// TIA Portal V17 export
// export: Created 2024-09-02T12:50:08.0346028Z, ExportSetting WithDefaults, DisplayName Totally Integrated Automation Portal, DisplayVersion V17, DisplayName TIA Portal Openness, DisplayVersion V17, DisplayName TIA Portal Version Control Interface, DisplayVersion V17, DisplayName STEP 7 Professional, DisplayVersion V17, DisplayName STEP 7 Safety, DisplayVersion V17, DisplayName WinCC Professional, DisplayVersion V17
FUNCTION "AnwFC1_FG02_Transport_OP70" : Void   // FC1381, LAD
TITLE = Transport
{ S7_Optimized_Access := 'TRUE' }
AUTHOR : VAF
FAMILY : SK
NAME : SK
VERSION : 0.1
// stored: AutoNumber false, IsIECCheckEnabled false, SetENOAutomatically false, UDAEnableTagReadback false
   VAR_TEMP
      Motion_Release : Bool;   // Bewegungsfreigabe / Motion permit
      Hand : Bool;
      Auto : Bool;
      t_ParityFault : Bool;
      t_ConfigFault : Bool;
      t_retval : Bool;
      "MM50/51_Home" : Bool;
      "MM50/51_Work" : Bool;
      "MM70/71_Home" : Bool;
      "MM70/71_Work" : Bool;
   END_VAR
BEGIN

REGION Network 1: Motion permit / Hand/ Auto / Bewegungsfreigabe / Hand / Auto
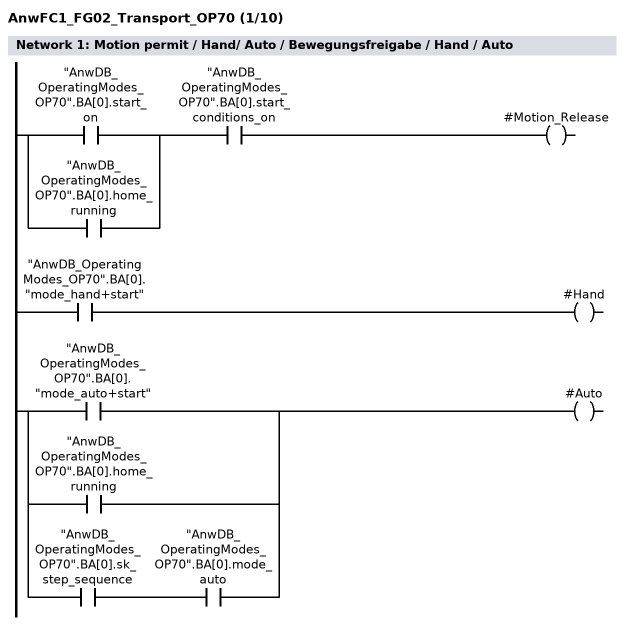
   RUNG wire#powerrail
      Contact( "AnwDB_OperatingModes_OP70".BA[0].start_on )
      wire#w1
      Contact( "AnwDB_OperatingModes_OP70".BA[0].start_conditions_on )
      Coil( #Motion_Release )
   END_RUNG
   RUNG wire#powerrail
      Contact( "AnwDB_OperatingModes_OP70".BA[0].home_running )
   END_RUNG wire#w1
   RUNG wire#powerrail
      Contact( "AnwDB_OperatingModes_OP70".BA[0]."mode_hand+start" )
      Coil( #Hand )
   END_RUNG
   RUNG wire#powerrail
      Contact( "AnwDB_OperatingModes_OP70".BA[0]."mode_auto+start" )
      wire#w2
      Coil( #Auto )
   END_RUNG
   RUNG wire#powerrail
      Contact( "AnwDB_OperatingModes_OP70".BA[0].home_running )
   END_RUNG wire#w2
   RUNG wire#powerrail
      Contact( "AnwDB_OperatingModes_OP70".BA[0].sk_step_sequence )
      Contact( "AnwDB_OperatingModes_OP70".BA[0].mode_auto )
   END_RUNG wire#w2
   // the same network as SCL:
   #Motion_Release := ("AnwDB_OperatingModes_OP70".BA[0].start_on OR "AnwDB_OperatingModes_OP70".BA[0].home_running) AND "AnwDB_OperatingModes_OP70".BA[0].start_conditions_on;
   #Hand := "AnwDB_OperatingModes_OP70".BA[0]."mode_hand+start";
   #Auto := "AnwDB_OperatingModes_OP70".BA[0]."mode_auto+start" OR "AnwDB_OperatingModes_OP70".BA[0].home_running OR ("AnwDB_OperatingModes_OP70".BA[0].sk_step_sequence AND "AnwDB_OperatingModes_OP70".BA[0].mode_auto);
END_REGION

REGION Network 2: Call of the step sequence / Aufruf der Schrittkette
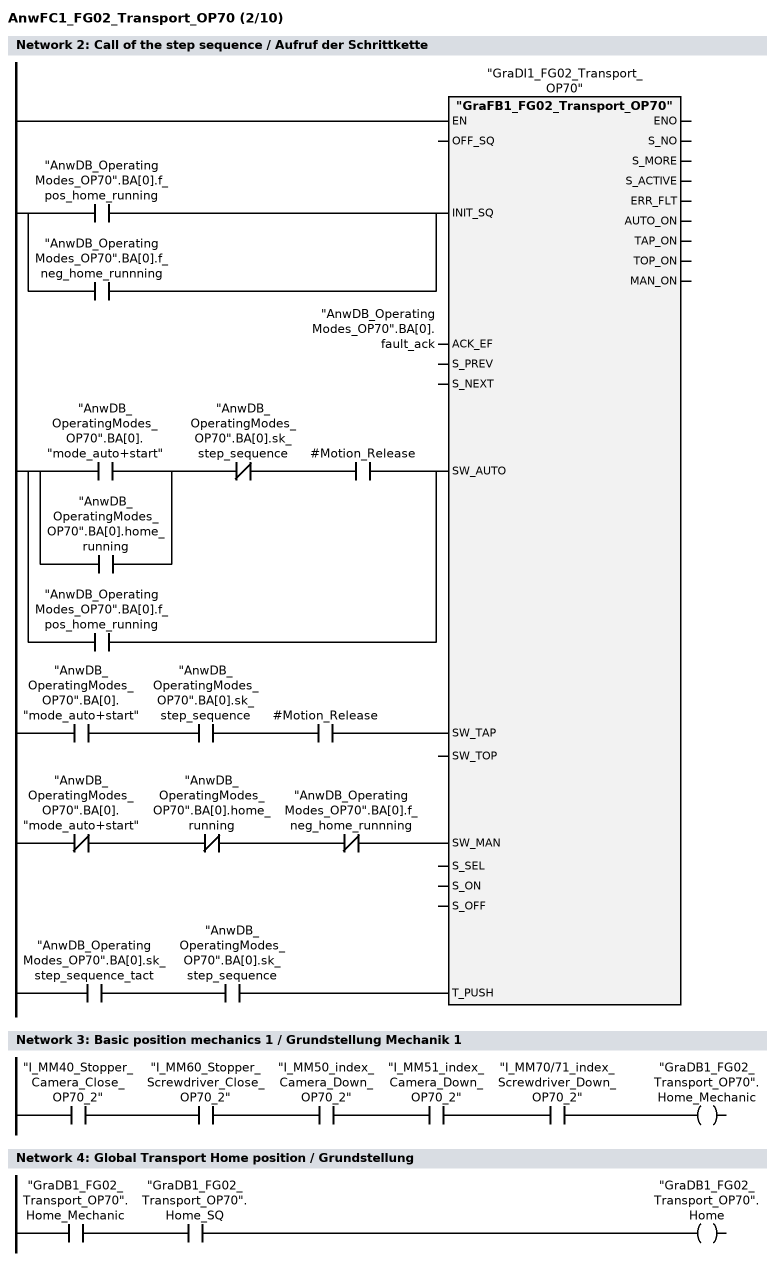
   RUNG wire#powerrail
      "GraDI1_FG02_Transport_OP70"(INIT_SQ := wire#w1, SW_AUTO := wire#w3, SW_TAP := wire#w4, SW_MAN := wire#w5, T_PUSH := wire#w6, OFF_SQ :=, ACK_EF := "AnwDB_OperatingModes_OP70".BA[0].fault_ack, S_PREV :=, S_NEXT :=, SW_TOP :=, S_SEL :=, S_ON :=, S_OFF :=, S_NO =>, S_MORE =>, S_ACTIVE =>, ERR_FLT =>, AUTO_ON =>, TAP_ON =>, TOP_ON =>, MAN_ON =>)
   END_RUNG
   RUNG wire#powerrail
      Contact( "AnwDB_OperatingModes_OP70".BA[0].f_pos_home_running )
   END_RUNG wire#w1
   RUNG wire#powerrail
      Contact( "AnwDB_OperatingModes_OP70".BA[0].f_neg_home_runnning )
   END_RUNG wire#w1
   RUNG wire#powerrail
      Contact( "AnwDB_OperatingModes_OP70".BA[0]."mode_auto+start" )
      wire#w2
      I_Contact( "AnwDB_OperatingModes_OP70".BA[0].sk_step_sequence )
      Contact( #Motion_Release )
   END_RUNG wire#w3
   RUNG wire#powerrail
      Contact( "AnwDB_OperatingModes_OP70".BA[0].home_running )
   END_RUNG wire#w2
   RUNG wire#powerrail
      Contact( "AnwDB_OperatingModes_OP70".BA[0].f_pos_home_running )
   END_RUNG wire#w3
   RUNG wire#powerrail
      Contact( "AnwDB_OperatingModes_OP70".BA[0]."mode_auto+start" )
      Contact( "AnwDB_OperatingModes_OP70".BA[0].sk_step_sequence )
      Contact( #Motion_Release )
   END_RUNG wire#w4
   RUNG wire#powerrail
      I_Contact( "AnwDB_OperatingModes_OP70".BA[0]."mode_auto+start" )
      I_Contact( "AnwDB_OperatingModes_OP70".BA[0].home_running )
      I_Contact( "AnwDB_OperatingModes_OP70".BA[0].f_neg_home_runnning )
   END_RUNG wire#w5
   RUNG wire#powerrail
      Contact( "AnwDB_OperatingModes_OP70".BA[0].sk_step_sequence_tact )
      Contact( "AnwDB_OperatingModes_OP70".BA[0].sk_step_sequence )
   END_RUNG wire#w6
   // the same network as SCL:
   "GraDI1_FG02_Transport_OP70"(INIT_SQ := "AnwDB_OperatingModes_OP70".BA[0].f_pos_home_running OR "AnwDB_OperatingModes_OP70".BA[0].f_neg_home_runnning,   // "GraFB1_FG02_Transport_OP70"
                           ACK_EF := "AnwDB_OperatingModes_OP70".BA[0].fault_ack,
                           SW_AUTO := (("AnwDB_OperatingModes_OP70".BA[0]."mode_auto+start" OR "AnwDB_OperatingModes_OP70".BA[0].home_running) AND NOT "AnwDB_OperatingModes_OP70".BA[0].sk_step_sequence AND #Motion_Release) OR "AnwDB_OperatingModes_OP70".BA[0].f_pos_home_running,
                           SW_TAP := "AnwDB_OperatingModes_OP70".BA[0]."mode_auto+start" AND "AnwDB_OperatingModes_OP70".BA[0].sk_step_sequence AND #Motion_Release,
                           SW_MAN := NOT "AnwDB_OperatingModes_OP70".BA[0]."mode_auto+start" AND NOT "AnwDB_OperatingModes_OP70".BA[0].home_running AND NOT "AnwDB_OperatingModes_OP70".BA[0].f_neg_home_runnning,
                           T_PUSH := "AnwDB_OperatingModes_OP70".BA[0].sk_step_sequence_tact AND "AnwDB_OperatingModes_OP70".BA[0].sk_step_sequence);
END_REGION

REGION Network 3: Basic position mechanics 1 / Grundstellung Mechanik 1
   RUNG wire#powerrail
      Contact( "I_MM40_Stopper_Camera_Close_OP70_2" )
      Contact( "I_MM60_Stopper_Screwdriver_Close_OP70_2" )
      Contact( "I_MM50_index_Camera_Down_OP70_2" )
      Contact( "I_MM51_index_Camera_Down_OP70_2" )
      Contact( "I_MM70/71_index_Screwdriver_Down_OP70_2" )
      Coil( "GraDB1_FG02_Transport_OP70".Home_Mechanic )
   END_RUNG
   // the same network as SCL:
   "GraDB1_FG02_Transport_OP70".Home_Mechanic := "I_MM40_Stopper_Camera_Close_OP70_2" AND "I_MM60_Stopper_Screwdriver_Close_OP70_2" AND "I_MM50_index_Camera_Down_OP70_2" AND "I_MM51_index_Camera_Down_OP70_2" AND "I_MM70/71_index_Screwdriver_Down_OP70_2";
END_REGION

REGION Network 4: Global Transport Home position / Grundstellung
   RUNG wire#powerrail
      Contact( "GraDB1_FG02_Transport_OP70".Home_Mechanic )
      Contact( "GraDB1_FG02_Transport_OP70".Home_SQ )
      Coil( "GraDB1_FG02_Transport_OP70".Home )
   END_RUNG
   // the same network as SCL:
   "GraDB1_FG02_Transport_OP70".Home := "GraDB1_FG02_Transport_OP70".Home_Mechanic AND "GraDB1_FG02_Transport_OP70".Home_SQ;
END_REGION

REGION Network 5: Finished message OK Camera / Fertigmeldung OK
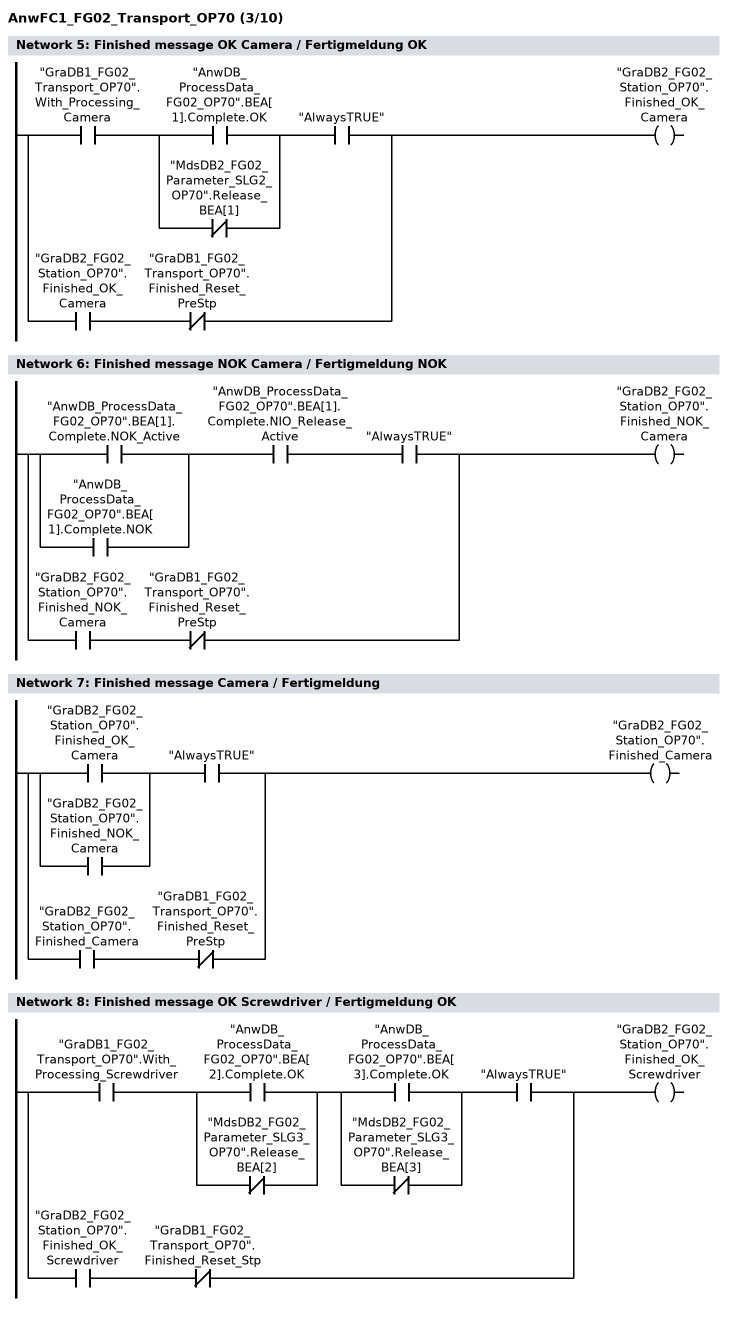
   RUNG wire#powerrail
      Contact( "GraDB1_FG02_Transport_OP70".With_Processing_Camera )
      wire#w1
      Contact( "AnwDB_ProcessData_FG02_OP70".BEA[1].Complete.OK )
      wire#w2
      Contact( "AlwaysTRUE" )
      wire#w3
      Coil( "GraDB2_FG02_Station_OP70".Finished_OK_Camera )
   END_RUNG
   RUNG wire#w1
      I_Contact( "MdsDB2_FG02_Parameter_SLG2_OP70".Release_BEA[1] )
   END_RUNG wire#w2
   RUNG wire#powerrail
      Contact( "GraDB2_FG02_Station_OP70".Finished_OK_Camera )
      I_Contact( "GraDB1_FG02_Transport_OP70".Finished_Reset_PreStp )
   END_RUNG wire#w3
   // the same network as SCL:
   "GraDB2_FG02_Station_OP70".Finished_OK_Camera := ("GraDB1_FG02_Transport_OP70".With_Processing_Camera AND ("AnwDB_ProcessData_FG02_OP70".BEA[1].Complete.OK OR NOT "MdsDB2_FG02_Parameter_SLG2_OP70".Release_BEA[1]) AND "AlwaysTRUE") OR ("GraDB2_FG02_Station_OP70".Finished_OK_Camera AND NOT "GraDB1_FG02_Transport_OP70".Finished_Reset_PreStp);
END_REGION

REGION Network 6: Finished message NOK Camera / Fertigmeldung NOK
   RUNG wire#powerrail
      Contact( "AnwDB_ProcessData_FG02_OP70".BEA[1].Complete.NOK_Active )
      wire#w1
      Contact( "AnwDB_ProcessData_FG02_OP70".BEA[1].Complete.NIO_Release_Active )
      Contact( "AlwaysTRUE" )
      wire#w2
      Coil( "GraDB2_FG02_Station_OP70".Finished_NOK_Camera )
   END_RUNG
   RUNG wire#powerrail
      Contact( "AnwDB_ProcessData_FG02_OP70".BEA[1].Complete.NOK )
   END_RUNG wire#w1
   RUNG wire#powerrail
      Contact( "GraDB2_FG02_Station_OP70".Finished_NOK_Camera )
      I_Contact( "GraDB1_FG02_Transport_OP70".Finished_Reset_PreStp )
   END_RUNG wire#w2
   // the same network as SCL:
   "GraDB2_FG02_Station_OP70".Finished_NOK_Camera := (("AnwDB_ProcessData_FG02_OP70".BEA[1].Complete.NOK_Active OR "AnwDB_ProcessData_FG02_OP70".BEA[1].Complete.NOK) AND "AnwDB_ProcessData_FG02_OP70".BEA[1].Complete.NIO_Release_Active AND "AlwaysTRUE") OR ("GraDB2_FG02_Station_OP70".Finished_NOK_Camera AND NOT "GraDB1_FG02_Transport_OP70".Finished_Reset_PreStp);
END_REGION

REGION Network 7: Finished message Camera / Fertigmeldung
   RUNG wire#powerrail
      Contact( "GraDB2_FG02_Station_OP70".Finished_OK_Camera )
      wire#w1
      Contact( "AlwaysTRUE" )
      wire#w2
      Coil( "GraDB2_FG02_Station_OP70".Finished_Camera )
   END_RUNG
   RUNG wire#powerrail
      Contact( "GraDB2_FG02_Station_OP70".Finished_NOK_Camera )
   END_RUNG wire#w1
   RUNG wire#powerrail
      Contact( "GraDB2_FG02_Station_OP70".Finished_Camera )
      I_Contact( "GraDB1_FG02_Transport_OP70".Finished_Reset_PreStp )
   END_RUNG wire#w2
   // the same network as SCL:
   "GraDB2_FG02_Station_OP70".Finished_Camera := (("GraDB2_FG02_Station_OP70".Finished_OK_Camera OR "GraDB2_FG02_Station_OP70".Finished_NOK_Camera) AND "AlwaysTRUE") OR ("GraDB2_FG02_Station_OP70".Finished_Camera AND NOT "GraDB1_FG02_Transport_OP70".Finished_Reset_PreStp);
END_REGION

REGION Network 8: Finished message OK Screwdriver / Fertigmeldung OK
   RUNG wire#powerrail
      Contact( "GraDB1_FG02_Transport_OP70".With_Processing_Screwdriver )
      wire#w1
      Contact( "AnwDB_ProcessData_FG02_OP70".BEA[2].Complete.OK )
      wire#w2
      Contact( "AnwDB_ProcessData_FG02_OP70".BEA[3].Complete.OK )
      wire#w3
      Contact( "AlwaysTRUE" )
      wire#w4
      Coil( "GraDB2_FG02_Station_OP70".Finished_OK_Screwdriver )
   END_RUNG
   RUNG wire#w1
      I_Contact( "MdsDB2_FG02_Parameter_SLG3_OP70".Release_BEA[2] )
   END_RUNG wire#w2
   RUNG wire#w2
      I_Contact( "MdsDB2_FG02_Parameter_SLG3_OP70".Release_BEA[3] )
   END_RUNG wire#w3
   RUNG wire#powerrail
      Contact( "GraDB2_FG02_Station_OP70".Finished_OK_Screwdriver )
      I_Contact( "GraDB1_FG02_Transport_OP70".Finished_Reset_Stp )
   END_RUNG wire#w4
   // the same network as SCL:
   "GraDB2_FG02_Station_OP70".Finished_OK_Screwdriver := ("GraDB1_FG02_Transport_OP70".With_Processing_Screwdriver AND ("AnwDB_ProcessData_FG02_OP70".BEA[2].Complete.OK OR NOT "MdsDB2_FG02_Parameter_SLG3_OP70".Release_BEA[2]) AND ("AnwDB_ProcessData_FG02_OP70".BEA[3].Complete.OK OR NOT "MdsDB2_FG02_Parameter_SLG3_OP70".Release_BEA[3]) AND "AlwaysTRUE") OR ("GraDB2_FG02_Station_OP70".Finished_OK_Screwdriver AND NOT "GraDB1_FG02_Transport_OP70".Finished_Reset_Stp);
END_REGION

REGION Network 9: Finished message NOK Screwdriver / Fertigmeldung NOK
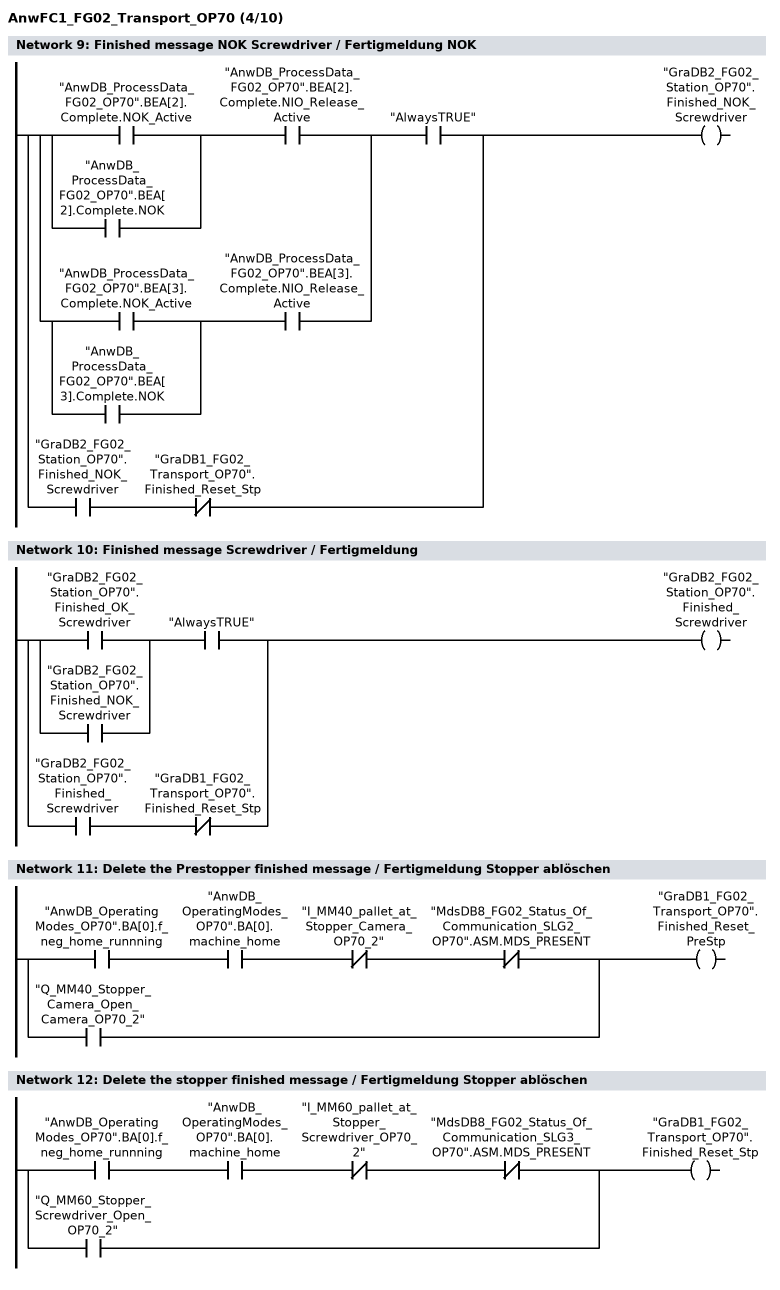
   RUNG wire#powerrail
      Contact( "AnwDB_ProcessData_FG02_OP70".BEA[2].Complete.NOK_Active )
      wire#w1
      Contact( "AnwDB_ProcessData_FG02_OP70".BEA[2].Complete.NIO_Release_Active )
      wire#w2
      Contact( "AlwaysTRUE" )
      wire#w4
      Coil( "GraDB2_FG02_Station_OP70".Finished_NOK_Screwdriver )
   END_RUNG
   RUNG wire#powerrail
      Contact( "AnwDB_ProcessData_FG02_OP70".BEA[2].Complete.NOK )
   END_RUNG wire#w1
   RUNG wire#powerrail
      Contact( "AnwDB_ProcessData_FG02_OP70".BEA[3].Complete.NOK_Active )
      wire#w3
      Contact( "AnwDB_ProcessData_FG02_OP70".BEA[3].Complete.NIO_Release_Active )
   END_RUNG wire#w2
   RUNG wire#powerrail
      Contact( "AnwDB_ProcessData_FG02_OP70".BEA[3].Complete.NOK )
   END_RUNG wire#w3
   RUNG wire#powerrail
      Contact( "GraDB2_FG02_Station_OP70".Finished_NOK_Screwdriver )
      I_Contact( "GraDB1_FG02_Transport_OP70".Finished_Reset_Stp )
   END_RUNG wire#w4
   // the same network as SCL:
   "GraDB2_FG02_Station_OP70".Finished_NOK_Screwdriver := (((("AnwDB_ProcessData_FG02_OP70".BEA[2].Complete.NOK_Active OR "AnwDB_ProcessData_FG02_OP70".BEA[2].Complete.NOK) AND "AnwDB_ProcessData_FG02_OP70".BEA[2].Complete.NIO_Release_Active) OR (("AnwDB_ProcessData_FG02_OP70".BEA[3].Complete.NOK_Active OR "AnwDB_ProcessData_FG02_OP70".BEA[3].Complete.NOK) AND "AnwDB_ProcessData_FG02_OP70".BEA[3].Complete.NIO_Release_Active)) AND "AlwaysTRUE") OR ("GraDB2_FG02_Station_OP70".Finished_NOK_Screwdriver AND NOT "GraDB1_FG02_Transport_OP70".Finished_Reset_Stp);
END_REGION

REGION Network 10: Finished message Screwdriver / Fertigmeldung
   RUNG wire#powerrail
      Contact( "GraDB2_FG02_Station_OP70".Finished_OK_Screwdriver )
      wire#w1
      Contact( "AlwaysTRUE" )
      wire#w2
      Coil( "GraDB2_FG02_Station_OP70".Finished_Screwdriver )
   END_RUNG
   RUNG wire#powerrail
      Contact( "GraDB2_FG02_Station_OP70".Finished_NOK_Screwdriver )
   END_RUNG wire#w1
   RUNG wire#powerrail
      Contact( "GraDB2_FG02_Station_OP70".Finished_Screwdriver )
      I_Contact( "GraDB1_FG02_Transport_OP70".Finished_Reset_Stp )
   END_RUNG wire#w2
   // the same network as SCL:
   "GraDB2_FG02_Station_OP70".Finished_Screwdriver := (("GraDB2_FG02_Station_OP70".Finished_OK_Screwdriver OR "GraDB2_FG02_Station_OP70".Finished_NOK_Screwdriver) AND "AlwaysTRUE") OR ("GraDB2_FG02_Station_OP70".Finished_Screwdriver AND NOT "GraDB1_FG02_Transport_OP70".Finished_Reset_Stp);
END_REGION

REGION Network 11: Delete the Prestopper finished message / Fertigmeldung Stopper ablöschen
   RUNG wire#powerrail
      Contact( "AnwDB_OperatingModes_OP70".BA[0].f_neg_home_runnning )
      Contact( "AnwDB_OperatingModes_OP70".BA[0].machine_home )
      I_Contact( "I_MM40_pallet_at_Stopper_Camera_OP70_2" )
      I_Contact( "MdsDB8_FG02_Status_Of_Communication_SLG2_OP70".ASM.MDS_PRESENT )
      wire#w1
      Coil( "GraDB1_FG02_Transport_OP70".Finished_Reset_PreStp )
   END_RUNG
   RUNG wire#powerrail
      Contact( "Q_MM40_Stopper_Camera_Open_Camera_OP70_2" )
   END_RUNG wire#w1
   // the same network as SCL:
   "GraDB1_FG02_Transport_OP70".Finished_Reset_PreStp := ("AnwDB_OperatingModes_OP70".BA[0].f_neg_home_runnning AND "AnwDB_OperatingModes_OP70".BA[0].machine_home AND NOT "I_MM40_pallet_at_Stopper_Camera_OP70_2" AND NOT "MdsDB8_FG02_Status_Of_Communication_SLG2_OP70".ASM.MDS_PRESENT) OR "Q_MM40_Stopper_Camera_Open_Camera_OP70_2";
END_REGION

REGION Network 12: Delete the stopper finished message / Fertigmeldung Stopper ablöschen
   RUNG wire#powerrail
      Contact( "AnwDB_OperatingModes_OP70".BA[0].f_neg_home_runnning )
      Contact( "AnwDB_OperatingModes_OP70".BA[0].machine_home )
      I_Contact( "I_MM60_pallet_at_Stopper_Screwdriver_OP70_2" )
      I_Contact( "MdsDB8_FG02_Status_Of_Communication_SLG3_OP70".ASM.MDS_PRESENT )
      wire#w1
      Coil( "GraDB1_FG02_Transport_OP70".Finished_Reset_Stp )
   END_RUNG
   RUNG wire#powerrail
      Contact( "Q_MM60_Stopper_Screwdriver_Open_OP70_2" )
   END_RUNG wire#w1
   // the same network as SCL:
   "GraDB1_FG02_Transport_OP70".Finished_Reset_Stp := ("AnwDB_OperatingModes_OP70".BA[0].f_neg_home_runnning AND "AnwDB_OperatingModes_OP70".BA[0].machine_home AND NOT "I_MM60_pallet_at_Stopper_Screwdriver_OP70_2" AND NOT "MdsDB8_FG02_Status_Of_Communication_SLG3_OP70".ASM.MDS_PRESENT) OR "Q_MM60_Stopper_Screwdriver_Open_OP70_2";
END_REGION

REGION Network 13: WT in Station
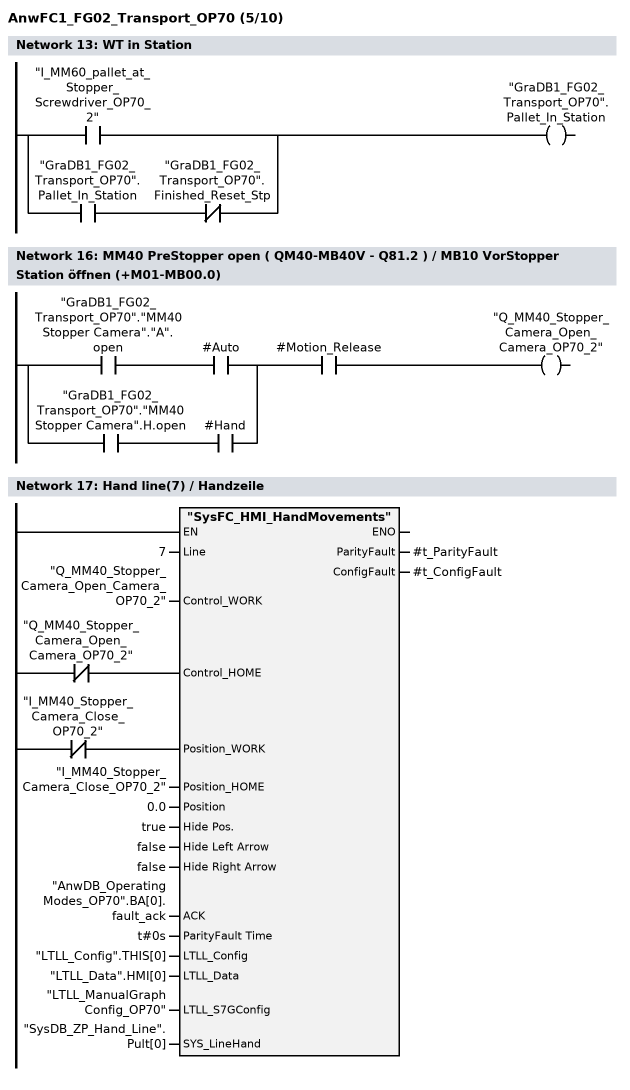
   RUNG wire#powerrail
      Contact( "I_MM60_pallet_at_Stopper_Screwdriver_OP70_2" )
      wire#w1
      Coil( "GraDB1_FG02_Transport_OP70".Pallet_In_Station )
   END_RUNG
   RUNG wire#powerrail
      Contact( "GraDB1_FG02_Transport_OP70".Pallet_In_Station )
      I_Contact( "GraDB1_FG02_Transport_OP70".Finished_Reset_Stp )
   END_RUNG wire#w1
   // the same network as SCL:
   "GraDB1_FG02_Transport_OP70".Pallet_In_Station := "I_MM60_pallet_at_Stopper_Screwdriver_OP70_2" OR ("GraDB1_FG02_Transport_OP70".Pallet_In_Station AND NOT "GraDB1_FG02_Transport_OP70".Finished_Reset_Stp);
END_REGION

REGION Network 14: ########### USER ########### / ########### ANWENDER ###########
END_REGION

REGION Network 15: ########### SS_02_001_Setup ###########
END_REGION

REGION Network 16: MM40 PreStopper open ( QM40-MB40V - Q81.2 ) / MB10 VorStopper Station öffnen (+M01-MB00.0)
   RUNG wire#powerrail
      Contact( "GraDB1_FG02_Transport_OP70"."MM40 Stopper Camera"."A".open )
      Contact( #Auto )
      wire#w1
      Contact( #Motion_Release )
      Coil( "Q_MM40_Stopper_Camera_Open_Camera_OP70_2" )
   END_RUNG
   RUNG wire#powerrail
      Contact( "GraDB1_FG02_Transport_OP70"."MM40 Stopper Camera".H.open )
      Contact( #Hand )
   END_RUNG wire#w1
   // the same network as SCL:
   "Q_MM40_Stopper_Camera_Open_Camera_OP70_2" := (("GraDB1_FG02_Transport_OP70"."MM40 Stopper Camera"."A".open AND #Auto) OR ("GraDB1_FG02_Transport_OP70"."MM40 Stopper Camera".H.open AND #Hand)) AND #Motion_Release;
END_REGION

REGION Network 17: Hand line(7) / Handzeile
   RUNG wire#powerrail
      "SysFC_HMI_HandMovements"(Control_HOME := wire#w1, Position_WORK := wire#w2, Line := 7, Control_WORK := "Q_MM40_Stopper_Camera_Open_Camera_OP70_2", Position_HOME := "I_MM40_Stopper_Camera_Close_OP70_2", Position := 0.0, "Hide Pos." := true, "Hide Left Arrow" := false, "Hide Right Arrow" := false, ACK := "AnwDB_OperatingModes_OP70".BA[0].fault_ack, "ParityFault Time" := t#0s, LTLL_Config := "LTLL_Config".THIS[0], LTLL_Data := "LTLL_Data".HMI[0], LTLL_S7GConfig := "LTLL_ManualGraphConfig_OP70", SYS_LineHand := "SysDB_ZP_Hand_Line".Pult[0], ParityFault => #t_ParityFault, ConfigFault => #t_ConfigFault)
   END_RUNG
   RUNG wire#powerrail
      I_Contact( "Q_MM40_Stopper_Camera_Open_Camera_OP70_2" )
   END_RUNG wire#w1
   RUNG wire#powerrail
      I_Contact( "I_MM40_Stopper_Camera_Close_OP70_2" )
   END_RUNG wire#w2
   // the same network as SCL:
   "SysFC_HMI_HandMovements"(Line := 7,
                           Control_WORK := "Q_MM40_Stopper_Camera_Open_Camera_OP70_2",
                           Control_HOME := NOT "Q_MM40_Stopper_Camera_Open_Camera_OP70_2",
                           Position_WORK := NOT "I_MM40_Stopper_Camera_Close_OP70_2",
                           Position_HOME := "I_MM40_Stopper_Camera_Close_OP70_2",
                           Position := 0.0,
                           "Hide Pos." := true,
                           "Hide Left Arrow" := false,
                           "Hide Right Arrow" := false,
                           ACK := "AnwDB_OperatingModes_OP70".BA[0].fault_ack,
                           "ParityFault Time" := t#0s,
                           LTLL_Config := "LTLL_Config".THIS[0],
                           LTLL_Data := "LTLL_Data".HMI[0],
                           LTLL_S7GConfig := "LTLL_ManualGraphConfig_OP70",
                           SYS_LineHand := "SysDB_ZP_Hand_Line".Pult[0],
                           ParityFault => #t_ParityFault,
                           ConfigFault => #t_ConfigFault);
END_REGION

REGION Network 18: Hand line SLG2 Prestopper read / write (8) / SLG BX600 schreiben / lesen
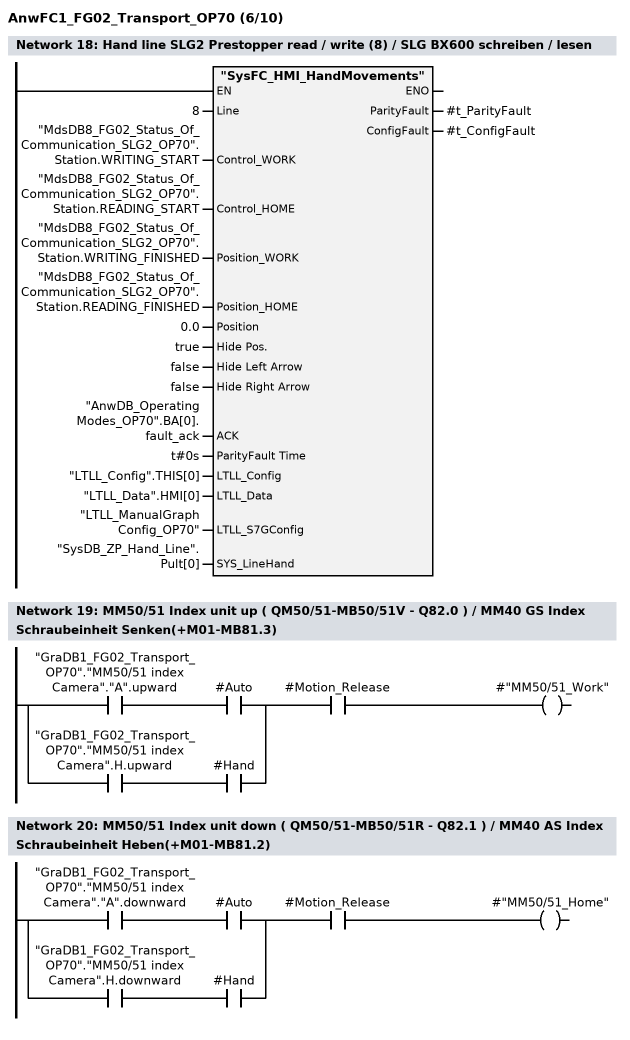
   RUNG wire#powerrail
      "SysFC_HMI_HandMovements"(Line := 8, Control_WORK := "MdsDB8_FG02_Status_Of_Communication_SLG2_OP70".Station.WRITING_START, Control_HOME := "MdsDB8_FG02_Status_Of_Communication_SLG2_OP70".Station.READING_START, Position_WORK := "MdsDB8_FG02_Status_Of_Communication_SLG2_OP70".Station.WRITING_FINISHED, Position_HOME := "MdsDB8_FG02_Status_Of_Communication_SLG2_OP70".Station.READING_FINISHED, Position := 0.0, "Hide Pos." := true, "Hide Left Arrow" := false, "Hide Right Arrow" := false, ACK := "AnwDB_OperatingModes_OP70".BA[0].fault_ack, "ParityFault Time" := t#0s, LTLL_Config := "LTLL_Config".THIS[0], LTLL_Data := "LTLL_Data".HMI[0], LTLL_S7GConfig := "LTLL_ManualGraphConfig_OP70", SYS_LineHand := "SysDB_ZP_Hand_Line".Pult[0], ParityFault => #t_ParityFault, ConfigFault => #t_ConfigFault)
   END_RUNG
   // the same network as SCL:
   "SysFC_HMI_HandMovements"(Line := 8,
                           Control_WORK := "MdsDB8_FG02_Status_Of_Communication_SLG2_OP70".Station.WRITING_START,
                           Control_HOME := "MdsDB8_FG02_Status_Of_Communication_SLG2_OP70".Station.READING_START,
                           Position_WORK := "MdsDB8_FG02_Status_Of_Communication_SLG2_OP70".Station.WRITING_FINISHED,
                           Position_HOME := "MdsDB8_FG02_Status_Of_Communication_SLG2_OP70".Station.READING_FINISHED,
                           Position := 0.0,
                           "Hide Pos." := true,
                           "Hide Left Arrow" := false,
                           "Hide Right Arrow" := false,
                           ACK := "AnwDB_OperatingModes_OP70".BA[0].fault_ack,
                           "ParityFault Time" := t#0s,
                           LTLL_Config := "LTLL_Config".THIS[0],
                           LTLL_Data := "LTLL_Data".HMI[0],
                           LTLL_S7GConfig := "LTLL_ManualGraphConfig_OP70",
                           SYS_LineHand := "SysDB_ZP_Hand_Line".Pult[0],
                           ParityFault => #t_ParityFault,
                           ConfigFault => #t_ConfigFault);
END_REGION

REGION Network 19: MM50/51 Index unit up ( QM50/51-MB50/51V - Q82.0 ) / MM40 GS Index Schraubeinheit Senken(+M01-MB81.3)
   RUNG wire#powerrail
      Contact( "GraDB1_FG02_Transport_OP70"."MM50/51 index Camera"."A".upward )
      Contact( #Auto )
      wire#w1
      Contact( #Motion_Release )
      Coil( #"MM50/51_Work" )
   END_RUNG
   RUNG wire#powerrail
      Contact( "GraDB1_FG02_Transport_OP70"."MM50/51 index Camera".H.upward )
      Contact( #Hand )
   END_RUNG wire#w1
   // the same network as SCL:
   #"MM50/51_Work" := (("GraDB1_FG02_Transport_OP70"."MM50/51 index Camera"."A".upward AND #Auto) OR ("GraDB1_FG02_Transport_OP70"."MM50/51 index Camera".H.upward AND #Hand)) AND #Motion_Release;
END_REGION

REGION Network 20: MM50/51 Index unit down ( QM50/51-MB50/51R - Q82.1 ) / MM40 AS Index Schraubeinheit Heben(+M01-MB81.2)
   RUNG wire#powerrail
      Contact( "GraDB1_FG02_Transport_OP70"."MM50/51 index Camera"."A".downward )
      Contact( #Auto )
      wire#w1
      Contact( #Motion_Release )
      Coil( #"MM50/51_Home" )
   END_RUNG
   RUNG wire#powerrail
      Contact( "GraDB1_FG02_Transport_OP70"."MM50/51 index Camera".H.downward )
      Contact( #Hand )
   END_RUNG wire#w1
   // the same network as SCL:
   #"MM50/51_Home" := (("GraDB1_FG02_Transport_OP70"."MM50/51 index Camera"."A".downward AND #Auto) OR ("GraDB1_FG02_Transport_OP70"."MM50/51 index Camera".H.downward AND #Hand)) AND #Motion_Release;
END_REGION

REGION Network 21: HLP - Index Up/Down / MM40 - HLP Pneumatik
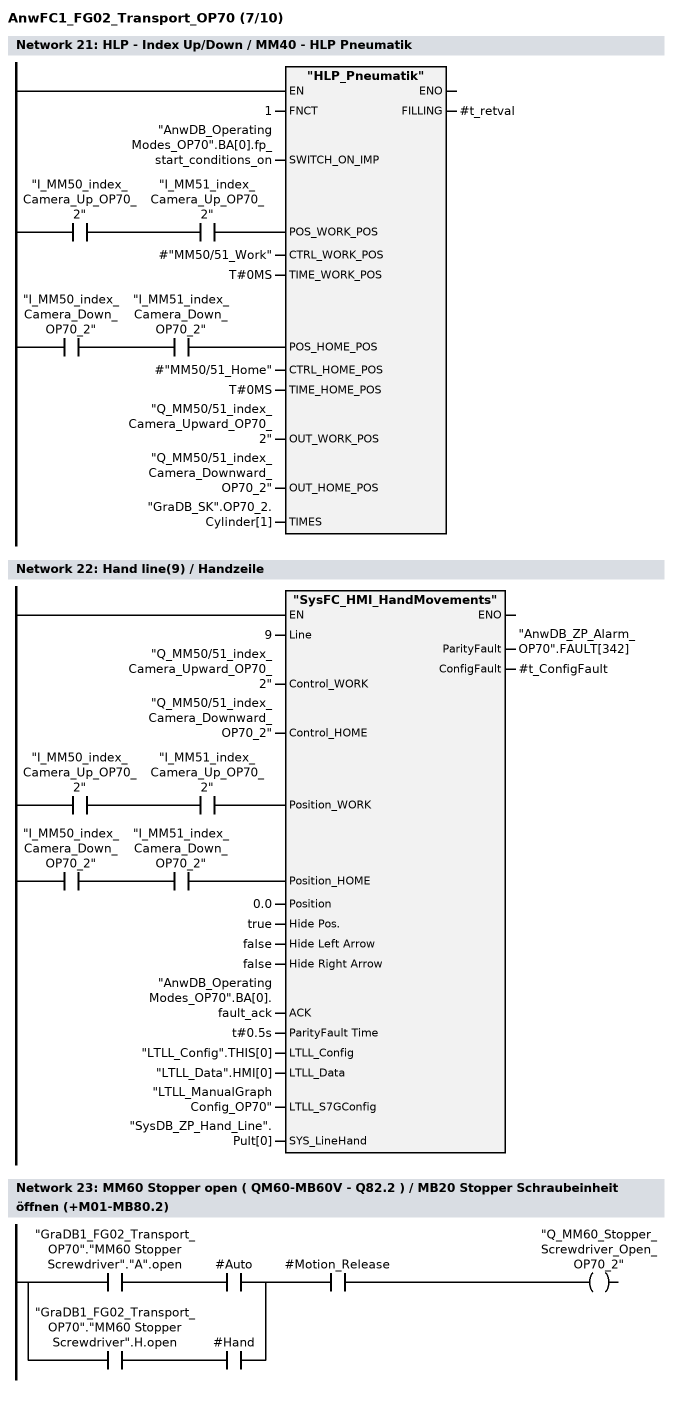
   RUNG wire#powerrail
      "HLP_Pneumatik"(POS_WORK_POS := wire#w1, POS_HOME_POS := wire#w2, FNCT := 1, SWITCH_ON_IMP := "AnwDB_OperatingModes_OP70".BA[0].fp_start_conditions_on, CTRL_WORK_POS := #"MM50/51_Work", TIME_WORK_POS := T#0MS, CTRL_HOME_POS := #"MM50/51_Home", TIME_HOME_POS := T#0MS, OUT_WORK_POS := "Q_MM50/51_index_Camera_Upward_OP70_2", OUT_HOME_POS := "Q_MM50/51_index_Camera_Downward_OP70_2", TIMES := "GraDB_SK".OP70_2.Cylinder[1], FILLING => #t_retval)
   END_RUNG
   RUNG wire#powerrail
      Contact( "I_MM50_index_Camera_Up_OP70_2" )
      Contact( "I_MM51_index_Camera_Up_OP70_2" )
   END_RUNG wire#w1
   RUNG wire#powerrail
      Contact( "I_MM50_index_Camera_Down_OP70_2" )
      Contact( "I_MM51_index_Camera_Down_OP70_2" )
   END_RUNG wire#w2
   // the same network as SCL:
   "HLP_Pneumatik"(FNCT := 1,
                   SWITCH_ON_IMP := "AnwDB_OperatingModes_OP70".BA[0].fp_start_conditions_on,
                   POS_WORK_POS := "I_MM50_index_Camera_Up_OP70_2" AND "I_MM51_index_Camera_Up_OP70_2",
                   CTRL_WORK_POS := #"MM50/51_Work",
                   TIME_WORK_POS := T#0MS,
                   POS_HOME_POS := "I_MM50_index_Camera_Down_OP70_2" AND "I_MM51_index_Camera_Down_OP70_2",
                   CTRL_HOME_POS := #"MM50/51_Home",
                   TIME_HOME_POS := T#0MS,
                   OUT_WORK_POS := "Q_MM50/51_index_Camera_Upward_OP70_2",
                   OUT_HOME_POS := "Q_MM50/51_index_Camera_Downward_OP70_2",
                   TIMES := "GraDB_SK".OP70_2.Cylinder[1],
                   FILLING => #t_retval);
END_REGION

REGION Network 22: Hand line(9) / Handzeile
   RUNG wire#powerrail
      "SysFC_HMI_HandMovements"(Position_WORK := wire#w1, Position_HOME := wire#w2, Line := 9, Control_WORK := "Q_MM50/51_index_Camera_Upward_OP70_2", Control_HOME := "Q_MM50/51_index_Camera_Downward_OP70_2", Position := 0.0, "Hide Pos." := true, "Hide Left Arrow" := false, "Hide Right Arrow" := false, ACK := "AnwDB_OperatingModes_OP70".BA[0].fault_ack, "ParityFault Time" := t#0.5s, LTLL_Config := "LTLL_Config".THIS[0], LTLL_Data := "LTLL_Data".HMI[0], LTLL_S7GConfig := "LTLL_ManualGraphConfig_OP70", SYS_LineHand := "SysDB_ZP_Hand_Line".Pult[0], ParityFault => "AnwDB_ZP_Alarm_OP70".FAULT[342], ConfigFault => #t_ConfigFault)
   END_RUNG
   RUNG wire#powerrail
      Contact( "I_MM50_index_Camera_Up_OP70_2" )
      Contact( "I_MM51_index_Camera_Up_OP70_2" )
   END_RUNG wire#w1
   RUNG wire#powerrail
      Contact( "I_MM50_index_Camera_Down_OP70_2" )
      Contact( "I_MM51_index_Camera_Down_OP70_2" )
   END_RUNG wire#w2
   // the same network as SCL:
   "SysFC_HMI_HandMovements"(Line := 9,
                           Control_WORK := "Q_MM50/51_index_Camera_Upward_OP70_2",
                           Control_HOME := "Q_MM50/51_index_Camera_Downward_OP70_2",
                           Position_WORK := "I_MM50_index_Camera_Up_OP70_2" AND "I_MM51_index_Camera_Up_OP70_2",
                           Position_HOME := "I_MM50_index_Camera_Down_OP70_2" AND "I_MM51_index_Camera_Down_OP70_2",
                           Position := 0.0,
                           "Hide Pos." := true,
                           "Hide Left Arrow" := false,
                           "Hide Right Arrow" := false,
                           ACK := "AnwDB_OperatingModes_OP70".BA[0].fault_ack,
                           "ParityFault Time" := t#0.5s,
                           LTLL_Config := "LTLL_Config".THIS[0],
                           LTLL_Data := "LTLL_Data".HMI[0],
                           LTLL_S7GConfig := "LTLL_ManualGraphConfig_OP70",
                           SYS_LineHand := "SysDB_ZP_Hand_Line".Pult[0],
                           ParityFault => "AnwDB_ZP_Alarm_OP70".FAULT[342],
                           ConfigFault => #t_ConfigFault);
END_REGION

REGION Network 23: MM60 Stopper open ( QM60-MB60V - Q82.2 ) / MB20 Stopper Schraubeinheit öffnen (+M01-MB80.2)
   RUNG wire#powerrail
      Contact( "GraDB1_FG02_Transport_OP70"."MM60 Stopper Screwdriver"."A".open )
      Contact( #Auto )
      wire#w1
      Contact( #Motion_Release )
      Coil( "Q_MM60_Stopper_Screwdriver_Open_OP70_2" )
   END_RUNG
   RUNG wire#powerrail
      Contact( "GraDB1_FG02_Transport_OP70"."MM60 Stopper Screwdriver".H.open )
      Contact( #Hand )
   END_RUNG wire#w1
   // the same network as SCL:
   "Q_MM60_Stopper_Screwdriver_Open_OP70_2" := (("GraDB1_FG02_Transport_OP70"."MM60 Stopper Screwdriver"."A".open AND #Auto) OR ("GraDB1_FG02_Transport_OP70"."MM60 Stopper Screwdriver".H.open AND #Hand)) AND #Motion_Release;
END_REGION

REGION Network 24: Hand line(10) / Handzeile
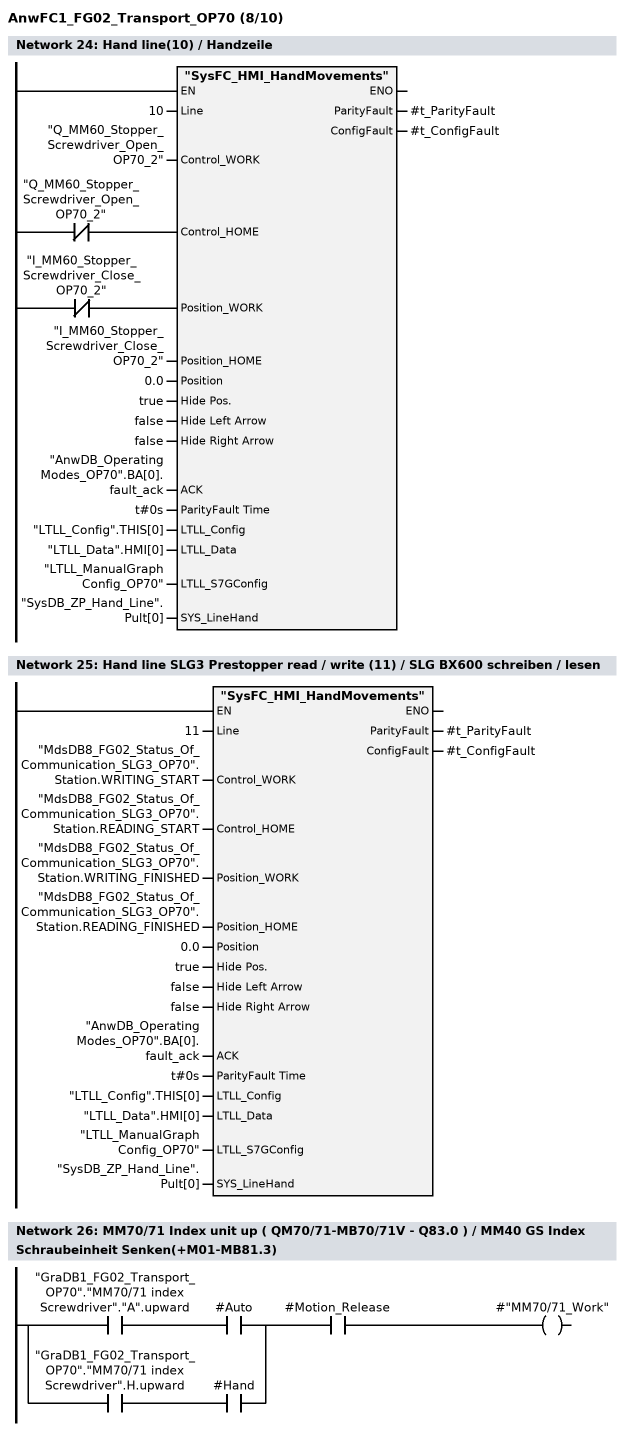
   RUNG wire#powerrail
      "SysFC_HMI_HandMovements"(Control_HOME := wire#w1, Position_WORK := wire#w2, Line := 10, Control_WORK := "Q_MM60_Stopper_Screwdriver_Open_OP70_2", Position_HOME := "I_MM60_Stopper_Screwdriver_Close_OP70_2", Position := 0.0, "Hide Pos." := true, "Hide Left Arrow" := false, "Hide Right Arrow" := false, ACK := "AnwDB_OperatingModes_OP70".BA[0].fault_ack, "ParityFault Time" := t#0s, LTLL_Config := "LTLL_Config".THIS[0], LTLL_Data := "LTLL_Data".HMI[0], LTLL_S7GConfig := "LTLL_ManualGraphConfig_OP70", SYS_LineHand := "SysDB_ZP_Hand_Line".Pult[0], ParityFault => #t_ParityFault, ConfigFault => #t_ConfigFault)
   END_RUNG
   RUNG wire#powerrail
      I_Contact( "Q_MM60_Stopper_Screwdriver_Open_OP70_2" )
   END_RUNG wire#w1
   RUNG wire#powerrail
      I_Contact( "I_MM60_Stopper_Screwdriver_Close_OP70_2" )
   END_RUNG wire#w2
   // the same network as SCL:
   "SysFC_HMI_HandMovements"(Line := 10,
                           Control_WORK := "Q_MM60_Stopper_Screwdriver_Open_OP70_2",
                           Control_HOME := NOT "Q_MM60_Stopper_Screwdriver_Open_OP70_2",
                           Position_WORK := NOT "I_MM60_Stopper_Screwdriver_Close_OP70_2",
                           Position_HOME := "I_MM60_Stopper_Screwdriver_Close_OP70_2",
                           Position := 0.0,
                           "Hide Pos." := true,
                           "Hide Left Arrow" := false,
                           "Hide Right Arrow" := false,
                           ACK := "AnwDB_OperatingModes_OP70".BA[0].fault_ack,
                           "ParityFault Time" := t#0s,
                           LTLL_Config := "LTLL_Config".THIS[0],
                           LTLL_Data := "LTLL_Data".HMI[0],
                           LTLL_S7GConfig := "LTLL_ManualGraphConfig_OP70",
                           SYS_LineHand := "SysDB_ZP_Hand_Line".Pult[0],
                           ParityFault => #t_ParityFault,
                           ConfigFault => #t_ConfigFault);
END_REGION

REGION Network 25: Hand line SLG3 Prestopper read / write (11) / SLG BX600 schreiben / lesen
   RUNG wire#powerrail
      "SysFC_HMI_HandMovements"(Line := 11, Control_WORK := "MdsDB8_FG02_Status_Of_Communication_SLG3_OP70".Station.WRITING_START, Control_HOME := "MdsDB8_FG02_Status_Of_Communication_SLG3_OP70".Station.READING_START, Position_WORK := "MdsDB8_FG02_Status_Of_Communication_SLG3_OP70".Station.WRITING_FINISHED, Position_HOME := "MdsDB8_FG02_Status_Of_Communication_SLG3_OP70".Station.READING_FINISHED, Position := 0.0, "Hide Pos." := true, "Hide Left Arrow" := false, "Hide Right Arrow" := false, ACK := "AnwDB_OperatingModes_OP70".BA[0].fault_ack, "ParityFault Time" := t#0s, LTLL_Config := "LTLL_Config".THIS[0], LTLL_Data := "LTLL_Data".HMI[0], LTLL_S7GConfig := "LTLL_ManualGraphConfig_OP70", SYS_LineHand := "SysDB_ZP_Hand_Line".Pult[0], ParityFault => #t_ParityFault, ConfigFault => #t_ConfigFault)
   END_RUNG
   // the same network as SCL:
   "SysFC_HMI_HandMovements"(Line := 11,
                           Control_WORK := "MdsDB8_FG02_Status_Of_Communication_SLG3_OP70".Station.WRITING_START,
                           Control_HOME := "MdsDB8_FG02_Status_Of_Communication_SLG3_OP70".Station.READING_START,
                           Position_WORK := "MdsDB8_FG02_Status_Of_Communication_SLG3_OP70".Station.WRITING_FINISHED,
                           Position_HOME := "MdsDB8_FG02_Status_Of_Communication_SLG3_OP70".Station.READING_FINISHED,
                           Position := 0.0,
                           "Hide Pos." := true,
                           "Hide Left Arrow" := false,
                           "Hide Right Arrow" := false,
                           ACK := "AnwDB_OperatingModes_OP70".BA[0].fault_ack,
                           "ParityFault Time" := t#0s,
                           LTLL_Config := "LTLL_Config".THIS[0],
                           LTLL_Data := "LTLL_Data".HMI[0],
                           LTLL_S7GConfig := "LTLL_ManualGraphConfig_OP70",
                           SYS_LineHand := "SysDB_ZP_Hand_Line".Pult[0],
                           ParityFault => #t_ParityFault,
                           ConfigFault => #t_ConfigFault);
END_REGION

REGION Network 26: MM70/71 Index unit up ( QM70/71-MB70/71V - Q83.0 ) / MM40 GS Index Schraubeinheit Senken(+M01-MB81.3)
   RUNG wire#powerrail
      Contact( "GraDB1_FG02_Transport_OP70"."MM70/71 index Screwdriver"."A".upward )
      Contact( #Auto )
      wire#w1
      Contact( #Motion_Release )
      Coil( #"MM70/71_Work" )
   END_RUNG
   RUNG wire#powerrail
      Contact( "GraDB1_FG02_Transport_OP70"."MM70/71 index Screwdriver".H.upward )
      Contact( #Hand )
   END_RUNG wire#w1
   // the same network as SCL:
   #"MM70/71_Work" := (("GraDB1_FG02_Transport_OP70"."MM70/71 index Screwdriver"."A".upward AND #Auto) OR ("GraDB1_FG02_Transport_OP70"."MM70/71 index Screwdriver".H.upward AND #Hand)) AND #Motion_Release;
END_REGION

REGION Network 27: MM70/71 Index unit down ( QM70/71-MB70/71R - Q83.1 ) / MM40 AS Index Schraubeinheit Heben(+M01-MB81.2)
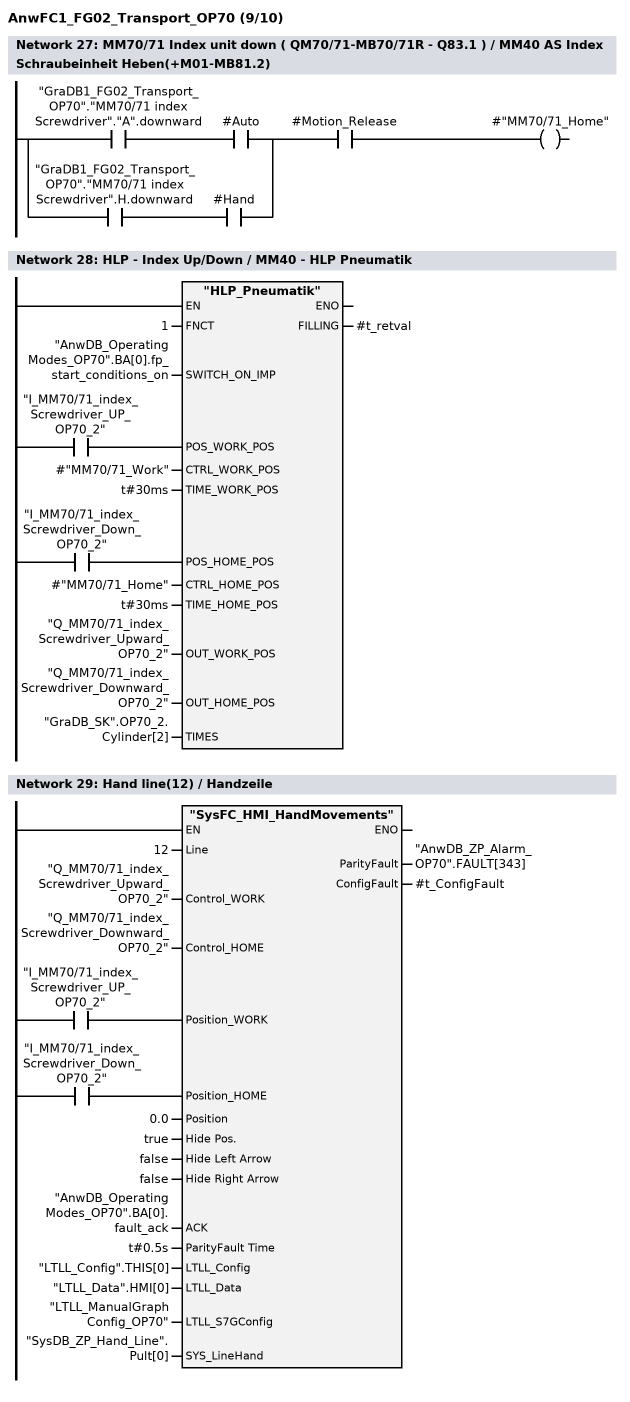
   RUNG wire#powerrail
      Contact( "GraDB1_FG02_Transport_OP70"."MM70/71 index Screwdriver"."A".downward )
      Contact( #Auto )
      wire#w1
      Contact( #Motion_Release )
      Coil( #"MM70/71_Home" )
   END_RUNG
   RUNG wire#powerrail
      Contact( "GraDB1_FG02_Transport_OP70"."MM70/71 index Screwdriver".H.downward )
      Contact( #Hand )
   END_RUNG wire#w1
   // the same network as SCL:
   #"MM70/71_Home" := (("GraDB1_FG02_Transport_OP70"."MM70/71 index Screwdriver"."A".downward AND #Auto) OR ("GraDB1_FG02_Transport_OP70"."MM70/71 index Screwdriver".H.downward AND #Hand)) AND #Motion_Release;
END_REGION

REGION Network 28: HLP - Index Up/Down / MM40 - HLP Pneumatik
   RUNG wire#powerrail
      "HLP_Pneumatik"(POS_WORK_POS := wire#w1, POS_HOME_POS := wire#w2, FNCT := 1, SWITCH_ON_IMP := "AnwDB_OperatingModes_OP70".BA[0].fp_start_conditions_on, CTRL_WORK_POS := #"MM70/71_Work", TIME_WORK_POS := t#30ms, CTRL_HOME_POS := #"MM70/71_Home", TIME_HOME_POS := t#30ms, OUT_WORK_POS := "Q_MM70/71_index_Screwdriver_Upward_OP70_2", OUT_HOME_POS := "Q_MM70/71_index_Screwdriver_Downward_OP70_2", TIMES := "GraDB_SK".OP70_2.Cylinder[2], FILLING => #t_retval)
   END_RUNG
   RUNG wire#powerrail
      Contact( "I_MM70/71_index_Screwdriver_UP_OP70_2" )
   END_RUNG wire#w1
   RUNG wire#powerrail
      Contact( "I_MM70/71_index_Screwdriver_Down_OP70_2" )
   END_RUNG wire#w2
   // the same network as SCL:
   "HLP_Pneumatik"(FNCT := 1,
                   SWITCH_ON_IMP := "AnwDB_OperatingModes_OP70".BA[0].fp_start_conditions_on,
                   POS_WORK_POS := "I_MM70/71_index_Screwdriver_UP_OP70_2",
                   CTRL_WORK_POS := #"MM70/71_Work",
                   TIME_WORK_POS := t#30ms,
                   POS_HOME_POS := "I_MM70/71_index_Screwdriver_Down_OP70_2",
                   CTRL_HOME_POS := #"MM70/71_Home",
                   TIME_HOME_POS := t#30ms,
                   OUT_WORK_POS := "Q_MM70/71_index_Screwdriver_Upward_OP70_2",
                   OUT_HOME_POS := "Q_MM70/71_index_Screwdriver_Downward_OP70_2",
                   TIMES := "GraDB_SK".OP70_2.Cylinder[2],
                   FILLING => #t_retval);
END_REGION

REGION Network 29: Hand line(12) / Handzeile
   RUNG wire#powerrail
      "SysFC_HMI_HandMovements"(Position_WORK := wire#w1, Position_HOME := wire#w2, Line := 12, Control_WORK := "Q_MM70/71_index_Screwdriver_Upward_OP70_2", Control_HOME := "Q_MM70/71_index_Screwdriver_Downward_OP70_2", Position := 0.0, "Hide Pos." := true, "Hide Left Arrow" := false, "Hide Right Arrow" := false, ACK := "AnwDB_OperatingModes_OP70".BA[0].fault_ack, "ParityFault Time" := t#0.5s, LTLL_Config := "LTLL_Config".THIS[0], LTLL_Data := "LTLL_Data".HMI[0], LTLL_S7GConfig := "LTLL_ManualGraphConfig_OP70", SYS_LineHand := "SysDB_ZP_Hand_Line".Pult[0], ParityFault => "AnwDB_ZP_Alarm_OP70".FAULT[343], ConfigFault => #t_ConfigFault)
   END_RUNG
   RUNG wire#powerrail
      Contact( "I_MM70/71_index_Screwdriver_UP_OP70_2" )
   END_RUNG wire#w1
   RUNG wire#powerrail
      Contact( "I_MM70/71_index_Screwdriver_Down_OP70_2" )
   END_RUNG wire#w2
   // the same network as SCL:
   "SysFC_HMI_HandMovements"(Line := 12,
                           Control_WORK := "Q_MM70/71_index_Screwdriver_Upward_OP70_2",
                           Control_HOME := "Q_MM70/71_index_Screwdriver_Downward_OP70_2",
                           Position_WORK := "I_MM70/71_index_Screwdriver_UP_OP70_2",
                           Position_HOME := "I_MM70/71_index_Screwdriver_Down_OP70_2",
                           Position := 0.0,
                           "Hide Pos." := true,
                           "Hide Left Arrow" := false,
                           "Hide Right Arrow" := false,
                           ACK := "AnwDB_OperatingModes_OP70".BA[0].fault_ack,
                           "ParityFault Time" := t#0.5s,
                           LTLL_Config := "LTLL_Config".THIS[0],
                           LTLL_Data := "LTLL_Data".HMI[0],
                           LTLL_S7GConfig := "LTLL_ManualGraphConfig_OP70",
                           SYS_LineHand := "SysDB_ZP_Hand_Line".Pult[0],
                           ParityFault => "AnwDB_ZP_Alarm_OP70".FAULT[343],
                           ConfigFault => #t_ConfigFault);
END_REGION

REGION Network 30: ##### Conveyors ON #####
END_REGION

REGION Network 31: Conveyor On
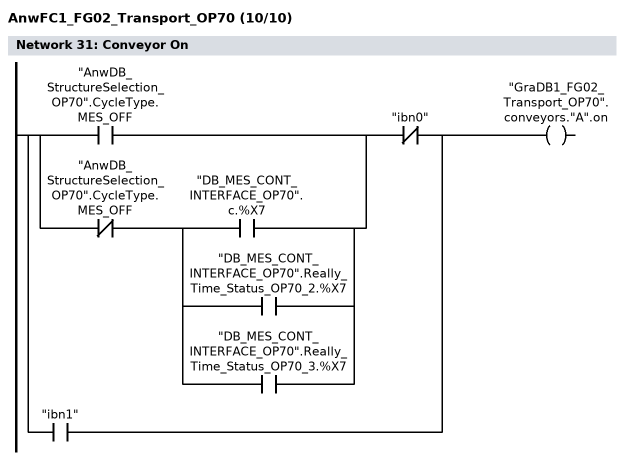
   RUNG wire#powerrail
      Contact( "AnwDB_StructureSelection_OP70".CycleType.MES_OFF )
      wire#w1
      I_Contact( "ibn0" )
      wire#w3
      Coil( "GraDB1_FG02_Transport_OP70".conveyors."A".on )
   END_RUNG
   RUNG wire#powerrail
      I_Contact( "AnwDB_StructureSelection_OP70".CycleType.MES_OFF )
      wire#w2
      Contact( "DB_MES_CONT_INTERFACE_OP70".c.%X7 )
   END_RUNG wire#w1
   RUNG wire#w2
      Contact( "DB_MES_CONT_INTERFACE_OP70".Really_Time_Status_OP70_2.%X7 )
   END_RUNG wire#w1
   RUNG wire#w2
      Contact( "DB_MES_CONT_INTERFACE_OP70".Really_Time_Status_OP70_3.%X7 )
   END_RUNG wire#w1
   RUNG wire#powerrail
      Contact( "ibn1" )
   END_RUNG wire#w3
   // the same network as SCL:
   "GraDB1_FG02_Transport_OP70".conveyors."A".on := (("AnwDB_StructureSelection_OP70".CycleType.MES_OFF OR (NOT "AnwDB_StructureSelection_OP70".CycleType.MES_OFF AND ("DB_MES_CONT_INTERFACE_OP70".c.%X7 OR "DB_MES_CONT_INTERFACE_OP70".Really_Time_Status_OP70_2.%X7 OR "DB_MES_CONT_INTERFACE_OP70".Really_Time_Status_OP70_3.%X7))) AND NOT "ibn0") OR "ibn1";
END_REGION
END_FUNCTION
